TYPE udtVFDCommand :
STRUCT
	Stop : BOOL;
	Start: BOOL;
	Jog: BOOL;
	ClearFaults: BOOL;
	RunFwd: BOOL;
	RunRev: BOOL;
	ForceKeypadCtrl: BOOL;
	MOPIncrement: BOOL;
	AccelRate1: BOOL;
	AccelRate2: BOOL;
	DecelRate1: BOOL;
	DecelRate2: BOOL;
	FreqSel01: BOOL;
	FreqSel02: BOOL;
	FreqSel03: BOOL;
	MOPDecrement: BOOL;
END_STRUCT
END_TYPE

(* stored: Version 1.1.0.1, ProductVersion 3.1.4020.12
   DUT udtVFDCommand: Id {5680323a-a88a-407d-b460-4c1303a14a92} *)
